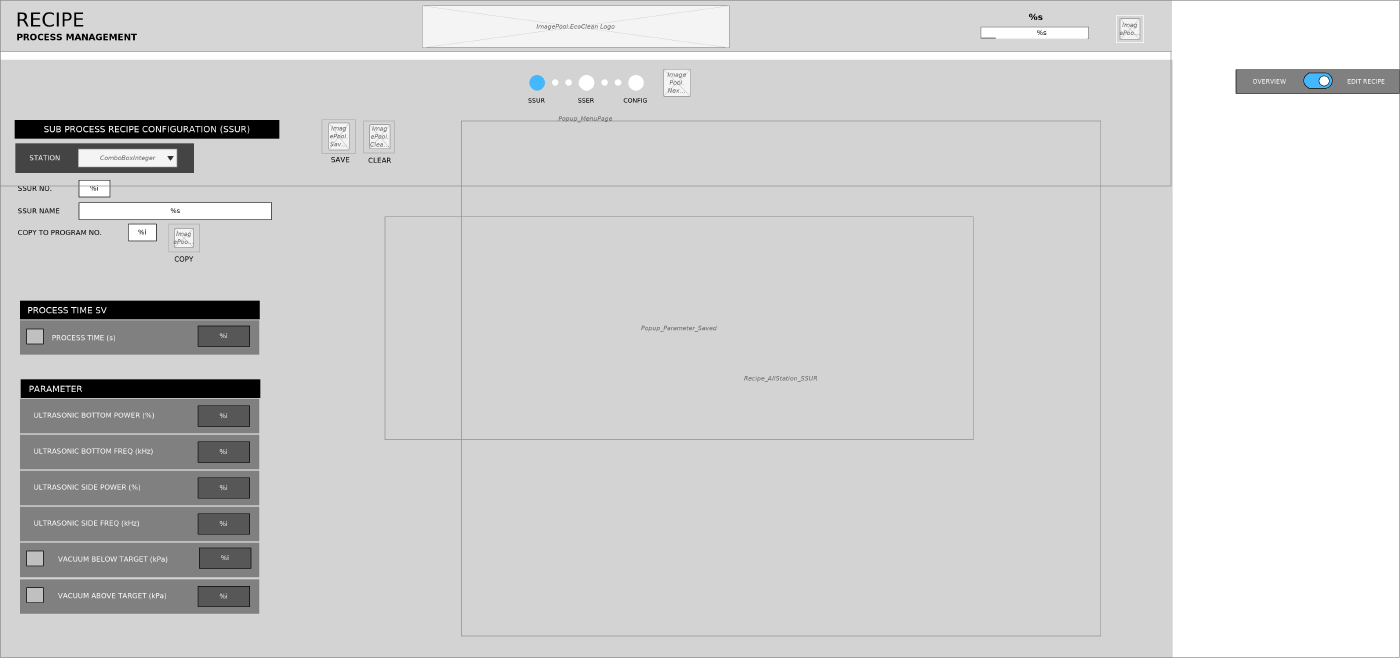
VISUALIZATION RecipeSSUR_Page  // 2293x1079
    Rectangle (0,98 1920x981)
    Rectangle (0,63 1920x26)
        p3528305787: HMI_Ctrl.ANIMATION3
    Rectangle (0,0 1919x85)
    Group (23,6 321x67)
        Label (0,0 267x53), "RECIPE"
        Label (1,43 320x24), "PROCESS MANAGEMENT"
    Frame (755,198 1048x845)
        shows Recipe_AllStation_SSUR()
    RoundedRectangle (25,235 292x48)
    Label (45,247 79x24), "STATION"
    Label (26,297 101x24), "SSUR NO."
    RoundedRectangle (129,295 51x28), "%i", text variable: DSScrMapSSUR.iSubRecipeNo
        OnMouseDown: write the text variable via VisuDialogs.Numpad, min 1, max 20
    Label (26,334 101x24), "SSUR NAME"
    RoundedRectangle (129,332 316x28), "%s", text variable: DSScrMapSSUR.sSubRecipeDescription
        OnMouseDown: write the text variable via VisuDialogs.Keypad
    Rectangle (24,197 433x30), "SUB PROCESS RECIPE CONFIGURATION (SSUR)"
    Label (26,361 156x41), "COPY TO PROGRAM NO."
    RoundedRectangle (210,367 46x28), "%i", text variable: DSScrMapSSUR.iCopyToSubRecipeNo
        OnMouseDown: write the text variable via VisuDialogs.Numpad, min 1, max 20
    ComboBoxInteger (128,244 162x30), variable: iStationNo, text list: 'TextList_Recipe'
    Group (1828,25 45x45)
        OnMouseClick: toggle HMI_Ctrl.MenuButton
        RoundedRectangle (0,0 45x45), colour toggle: HMI_Ctrl.MenuButton
        Image (6,5 33x35), image: ImagePool.Menu Button
    Group (2024,113 269x41)
        RoundedRectangle (0,1 269x39)
        Label (1,0 108x41), "OVERVIEW"
        Label (161,0 105x41), "EDIT RECIPE"
        Group (111,6 47x26)
            OnMouseClick: change screen: Recipe_Page
            Group (0,0 47x26)
                Ellipse (0,0 26x26)
                Ellipse (21,0 26x26)
                RoundedRectangle (8,0 29x26)
            Ellipse (1,1 24x24)
            Ellipse (23,1 23x24)
            RoundedRectangle (9,1 28x24)
            Ellipse (25,5 17x17)
    Ellipse (867,123 25x25)
    Ellipse (948,123 25x25)
    Ellipse (904,130 10x10)
    Ellipse (926,130 10x10)
    Ellipse (985,130 10x10)
    Ellipse (1007,130 10x10)
    Ellipse (1029,123 25x25)
    Label (847,153 64x24), "SSUR"
    Label (928,153 64x24), "SSER"
    Label (1009,153 64x24), "CONFIG"
    Image (1086,113 45x45), image: ImagePool.Next Button
        OnMouseClick: change screen: RecipeSSER_Page
    Rectangle (33,525 391x56)
    Label (82,546 150x16), "PROCESS TIME (s)"
    Rectangle (324,534 85x34), "%i", text variable: DSScrMapSSUR.DsSubRecipeMemory.iComCon5ProcessTimer, invisible if: NOT.DSScrMapSSUR.DsSubRecipeMemory.bComCon20EnProcessTimer
        OnMouseDown: write the text variable via VisuDialogs.Numpad, min 0, max 9999
    Rectangle (33,493 392x30)
    Label (42,501 304x16), "PROCESS TIME SV"
    Rectangle (43,539 28x25)
        toggle DSScrMapSSUR.DsSubRecipeMemory.bComCon20EnProcessTimer
    Label (46,719 150x16)
    Label (46,687 150x16)
    Rectangle (33,654 391x56), invisible if: NOT DSScrMapSSUR.DsSubRecipeMemory.bOut3EnProTankBottomUltrasonicA
    Label (52,673 240x16), "ULTRASONIC BOTTOM POWER (%)", invisible if: NOT DSScrMapSSUR.DsSubRecipeMemory.bOut3EnProTankBottomUltrasonicA
    Rectangle (324,665 85x34), "%i", text variable: DSScrMapSSUR.DsSubRecipeMemory.iOut3ProTankBtmUsAPwrPercent, invisible if: NOT DSScrMapSSUR.DsSubRecipeMemory.bOut3EnProTankBottomUltrasonicA
        OnMouseDown: write the text variable via VisuDialogs.Numpad, min 10, max 100
    Rectangle (33,713 391x56), invisible if: NOT DSScrMapSSUR.DsSubRecipeMemory.bOut3EnProTankBottomUltrasonicA
    Label (52,732 239x16), "ULTRASONIC BOTTOM FREQ (kHz)", invisible if: NOT DSScrMapSSUR.DsSubRecipeMemory.bOut3EnProTankBottomUltrasonicA
    Rectangle (324,724 85x34), "%i", text variable: .DSScrMapSSUR.DsSubRecipeMemory.iOut8ProTankBtmUsAkHz, invisible if: NOT DSScrMapSSUR.DsSubRecipeMemory.bOut3EnProTankBottomUltrasonicA
        tap bFreqBtmChange[iStationNo]
    Rectangle (34,622 392x30)
    Label (44,630 304x16), "PARAMETER"
    Image (691,9 504x69), image: ImagePool.EcoClean Logo
    Group (276,367 51x70), invisible if: bMainOnOff
        RoundedRectangle (0,0 51x46), colour toggle: DSScrMapSSUR.bCopyPB
            tap DSScrMapSSUR.bCopyPB
        Image (9,7 32x32), image: ImagePool.Copy Button
            OnMouseDown: execute { DSScrMapSSUR.bCopyPB:=1; }
            OnMouseUp: execute { DSScrMapSSUR.bCopyPB:=0; }
        Label (4,46 42x24), "COPY"
    Group (1606,17 179x46)
        Button (0,27 177x19), image: VisuSymbols.Symbols.AddUser
        Rectangle (25,28 150x18), "%s", text variable: fbHmiTF1800_UserlevelManagement.dsHmiUserStatus_Active.sLoginName
        Rectangle (2,0 177x22), "%s", text variable: DSLocalSystemTimeML.sCurrentDT24Hr_General
    Group (527,196 56x80), invisible if: bMainOnOff
        Label (5,52 51x28), "SAVE", invisible if: bMainOnOff
        RoundedRectangle (0,0 55x56), colour toggle: bRecipeSavePb
            tap bRecipeSavePb
        Image (11,5 34x45), image: ImagePool.Save Button
            OnMouseDown: execute { bRecipeSavePb:=1; }
            OnMouseUp: execute { bRecipeSavePb:=0; }
    Frame (630,355 964x366), invisible if: NOT stWritePersistentData.SaveHR
        shows Popup_Parameter_Saved()
    Rectangle (33,890 391x56), invisible if: iStationNo<>6 OR NOT DSScrMapSSUR.DsSubRecipeMemory.bOut11EnVacuumPump
    Label (92,909 221x16), "VACUUM BELOW TARGET (kPa)", invisible if: iStationNo<>6 OR NOT DSScrMapSSUR.DsSubRecipeMemory.bOut11EnVacuumPump
    Rectangle (326,898 85x34), "%i", text variable: DSScrMapSSUR.DsSubRecipeMemory.iComCon1TargetVacuumLevel, invisible if: NOT DSScrMapSSUR.DsSubRecipeMemory.bComCon11EnBelowTargetVacuumLevel
        OnMouseDown: write the text variable via VisuDialogs.Numpad, min -120, max 10
    Rectangle (33,950 391x56), invisible if: iStationNo<>6 OR NOT DSScrMapSSUR.DsSubRecipeMemory.bOut11EnVacuumPump
    Label (92,969 214x16), "VACUUM ABOVE TARGET (kPa)", invisible if: iStationNo<>6 OR NOT DSScrMapSSUR.DsSubRecipeMemory.bOut11EnVacuumPump
    Rectangle (324,961 85x34), "%i", text variable: DSScrMapSSUR.DsSubRecipeMemory.iComCon1TargetVacuumLevel, invisible if: NOT DSScrMapSSUR.DsSubRecipeMemory.bComCon12EnAboveTargetVacuumLevel
        OnMouseDown: write the text variable via VisuDialogs.Numpad, min -120, max 10
    Label (46,837 150x16)
    Label (46,805 150x16)
    Rectangle (33,772 391x56), invisible if: NOT DSScrMapSSUR.DsSubRecipeMemory.bOut6EnProTankSideUltrasonicA
    Label (52,791 212x16), "ULTRASONIC SIDE POWER (%)", invisible if: NOT DSScrMapSSUR.DsSubRecipeMemory.bOut6EnProTankSideUltrasonicA
    Rectangle (324,783 85x34), "%i", text variable: DSScrMapSSUR.DsSubRecipeMemory.iOut6ProTankSideUsAPwrPercent, invisible if: NOT DSScrMapSSUR.DsSubRecipeMemory.bOut6EnProTankSideUltrasonicA
        OnMouseDown: write the text variable via VisuDialogs.Numpad, min 10, max 100
    Rectangle (33,831 391x56), invisible if: NOT DSScrMapSSUR.DsSubRecipeMemory.bOut6EnProTankSideUltrasonicA
    Label (52,850 217x16), "ULTRASONIC SIDE FREQ (kHz)", invisible if: NOT DSScrMapSSUR.DsSubRecipeMemory.bOut6EnProTankSideUltrasonicA
    Rectangle (324,842 85x34), "%i", text variable: .DSScrMapSSUR.DsSubRecipeMemory.iOut11ProTankSideUsAkHz, invisible if: NOT DSScrMapSSUR.DsSubRecipeMemory.bOut6EnProTankSideUltrasonicA
        tap bFreqSideChange[iStationNo]
    Rectangle (43,903 28x25), invisible if: iStationNo<>6 OR NOT DSScrMapSSUR.DsSubRecipeMemory.bOut11EnVacuumPump
        toggle DSScrMapSSUR.DsSubRecipeMemory.bComCon11EnBelowTargetVacuumLevel
    Rectangle (43,963 28x25), invisible if: iStationNo<>6 OR NOT DSScrMapSSUR.DsSubRecipeMemory.bOut11EnVacuumPump
        toggle DSScrMapSSUR.DsSubRecipeMemory.bComCon12EnAboveTargetVacuumLevel
    RoundedRectangle (595,198 51x53), colour toggle: bRecipeClearInd_SSER
        tap bBufferClearPB_SSUR[iStationNo]
    Label (597,251 50x24), "CLEAR"
    Image (605,204 34x40), image: ImagePool.Clear Button
        OnMouseDown: execute { bBufferClearPB_SSUR[iStationNo]:=1; }
        OnMouseUp: execute { bBufferClearPB_SSUR[iStationNo]:=0; }
    Frame (0,84 1918x221), invisible if: HMI_Ctrl.CloseMenuButton
        shows Popup_MenuPage()
END_VISUALIZATION

(* stored: Version 1.1.0.1, ProductVersion 3.1.4024.12
   Visu RecipeSSUR_Page: Id {ceb1ba28-e51f-4e36-89a8-10c36669699d} *)
